INTERFACE IAngleSequenceOrientation

END_INTERFACE

(* stored: Version 1.1.0.1, ProductVersion 3.1.4024.9
   Itf IAngleSequenceOrientation: Id {8b8f642f-56a7-0e07-3314-3e8f93c5ace1} *)
